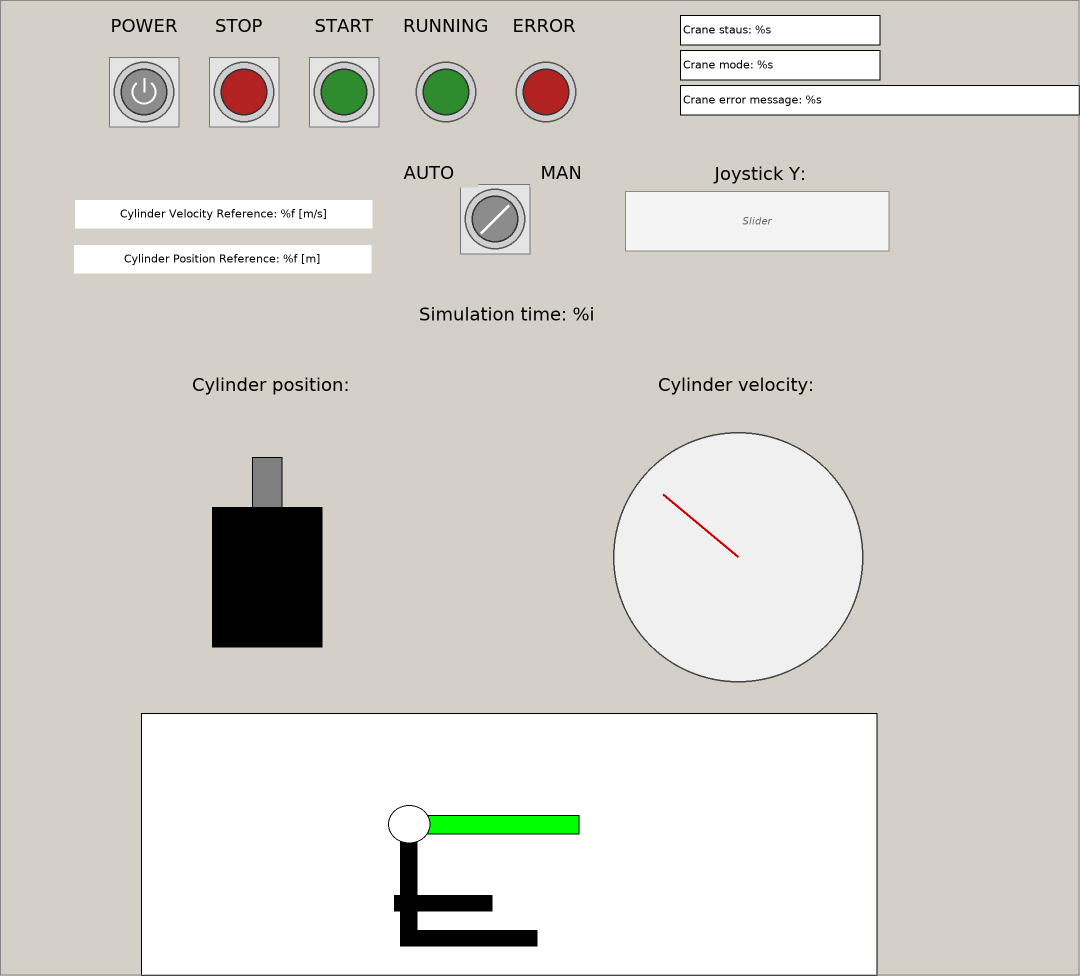
VISUALIZATION CraneSimulationHMI  // 1080x976
    PowerSwitch (109,57 70x70), variable: Inputs.bOnSelector, behaviour: TOGGLE, style: Switch-PowerSwitch-Gray
    RotarySwitch (460,184 70x70), variable: Inputs.bAutoSelector, behaviour: TOGGLE, style: Switch-RotarySwitch-Gray
    PushSwitch (309,57 70x70), variable: Inputs.bStartButton, behaviour: TOGGLE, style: Switch-PushSwitch-Green
    Rectangle (94,12 100x28), "POWER"
    Rectangle (294,12 100x28), "START"
    Rectangle (380,159 98x28), "AUTO"
    Rectangle (530,159 98x28), "MANUAL"
    Lamp1 (411,57 70x70), variable: Outputs.bStartLight, style: Lamp-Lamp1-Green
    Rectangle (396,12 100x28), "RUNNING"
    Rectangle (239,301 536x27), "Simulation time: %i", text variable: Parameters.stStateVariables.fTime
    Meter360 (613,432 250x250), value: HMI.fCylinderVelocity, style: Meter-Meter360-Gray, scale format: %.2f, scale -0.05..0.05
    Rectangle (182,372 178x26), "Cylinder position:"
    Rectangle (647,372 178x26), "Cylinder velocity:"
    Rectangle (680,85 400x30), "Crane error message: %s", text variable: HMI.sPistonEndStopMessage
    Rectangle (680,50 200x30), "Crane mode: %s", text variable: Outputs.eCraneMode
    Rectangle (680,15 200x30), "Crane staus: %s", text variable: Outputs.eCraneStatus
    Rectangle (252,457 30x180)
        p2738717112: -HMI.fCylinderPositon*100
    Rectangle (212,507 110x140)
    Textfield (73,244 299x30), "Cylinder Position Reference: %f [m]", text variable: HMI.fCylinderPositon
    Textfield (74,199 299x30), "Cylinder Velocity Reference: %f [m/s]", text variable: HMI.fCylinderVelocity
        OnMouseClick: write the text variable via Default
    PushSwitch (209,57 70x70), variable: Inputs.bStopButton, behaviour: TAP, style: Switch-PushSwitch-Red
    Rectangle (189,12 100x28), "STOP"
    Rectangle (141,713 736x263)
    Rectangle (400,930 137x16)
    Rectangle (400,810 17x130)
    Rectangle (409,815 170x19), angle 5
        p2858320360: -HMI.fBoomAngle
    Ellipse (388,805 42x38)
    Lamp1 (511,57 70x70), variable: Outputs.bStopLight, style: Lamp-Lamp1-Red
    Rectangle (494,12 100x28), "ERROR"
    Rectangle (394,895 98x16), angle 43
    Rectangle (580,162 361x24), "Joystick Y:"
    Slider (625,191 264x60), variable: Inputs.fJoystickY, scale -1..1
END_VISUALIZATION

(* stored: Version 1.1.0.1, ProductVersion 3.1.4024.10
   Visu CraneSimulationHMI: Id {b5520909-ac3e-4cb2-bbd3-14e4794d6a77} *)
